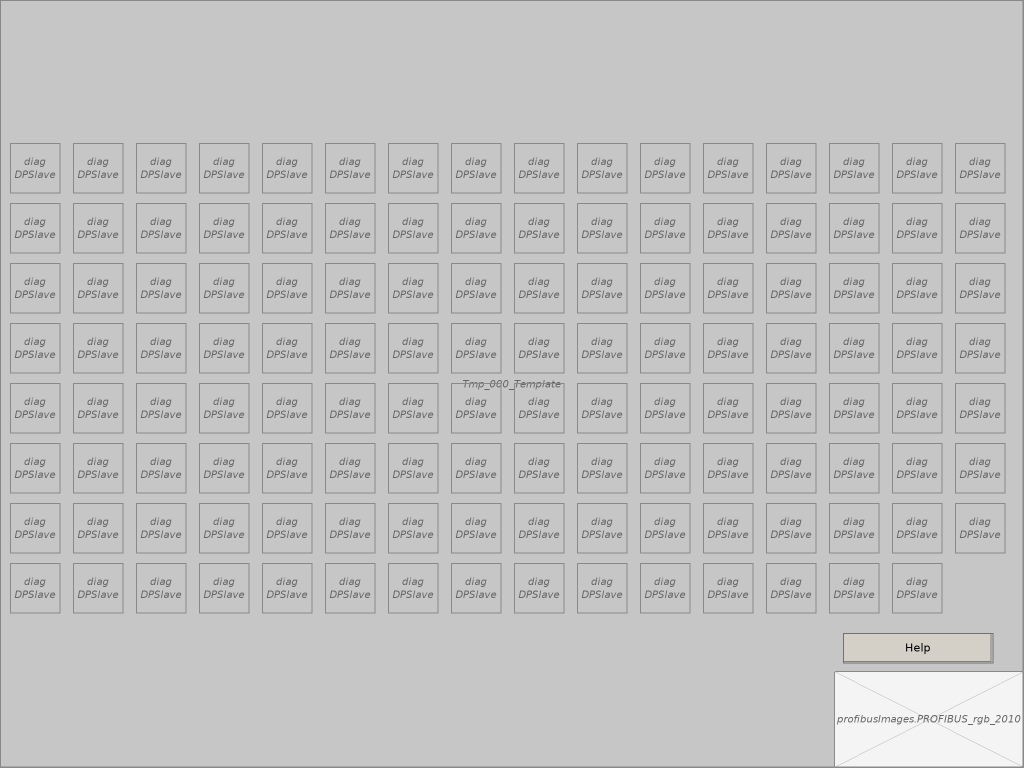
VISUALIZATION Dia_802_Profibus  // 1024x768
    Frame (0,0 1024x768)
        shows Tmp_000_Template(header := gHMIData.hmiHeader)
    Group (10,143 995x50)
        Frame (0,0 50x50)
            shows diagDPSlave(dataValues := profibusDiag.DPslaveDiag[1])
        Frame (63,0 50x50)
            shows diagDPSlave(dataValues := profibusDiag.DPslaveDiag[2])
        Frame (126,0 50x50)
            shows diagDPSlave(dataValues := profibusDiag.DPslaveDiag[3])
        Frame (189,0 50x50)
            shows diagDPSlave(dataValues := profibusDiag.DPslaveDiag[4])
        Frame (252,0 50x50)
            shows diagDPSlave(dataValues := profibusDiag.DPslaveDiag[5])
        Frame (315,0 50x50)
            shows diagDPSlave(dataValues := profibusDiag.DPslaveDiag[6])
        Frame (378,0 50x50)
            shows diagDPSlave(dataValues := profibusDiag.DPslaveDiag[7])
        Frame (441,0 50x50)
            shows diagDPSlave(dataValues := profibusDiag.DPslaveDiag[8])
        Frame (504,0 50x50)
            shows diagDPSlave(dataValues := profibusDiag.DPslaveDiag[9])
        Frame (567,0 50x50)
            shows diagDPSlave(dataValues := profibusDiag.DPslaveDiag[10])
        Frame (630,0 50x50)
            shows diagDPSlave(dataValues := profibusDiag.DPslaveDiag[11])
        Frame (693,0 50x50)
            shows diagDPSlave(dataValues := profibusDiag.DPslaveDiag[12])
        Frame (756,0 50x50)
            shows diagDPSlave(dataValues := profibusDiag.DPslaveDiag[13])
        Frame (819,0 50x50)
            shows diagDPSlave(dataValues := profibusDiag.DPslaveDiag[14])
        Frame (882,0 50x50)
            shows diagDPSlave(dataValues := profibusDiag.DPslaveDiag[15])
        Frame (945,0 50x50)
            shows diagDPSlave(dataValues := profibusDiag.DPslaveDiag[16])
    Group (10,203 995x50)
        Frame (0,0 50x50)
            shows diagDPSlave(dataValues := profibusDiag.DPslaveDiag[17])
        Frame (63,0 50x50)
            shows diagDPSlave(dataValues := profibusDiag.DPslaveDiag[18])
        Frame (126,0 50x50)
            shows diagDPSlave(dataValues := profibusDiag.DPslaveDiag[19])
        Frame (189,0 50x50)
            shows diagDPSlave(dataValues := profibusDiag.DPslaveDiag[20])
        Frame (252,0 50x50)
            shows diagDPSlave(dataValues := profibusDiag.DPslaveDiag[21])
        Frame (315,0 50x50)
            shows diagDPSlave(dataValues := profibusDiag.DPslaveDiag[22])
        Frame (378,0 50x50)
            shows diagDPSlave(dataValues := profibusDiag.DPslaveDiag[23])
        Frame (441,0 50x50)
            shows diagDPSlave(dataValues := profibusDiag.DPslaveDiag[24])
        Frame (504,0 50x50)
            shows diagDPSlave(dataValues := profibusDiag.DPslaveDiag[25])
        Frame (567,0 50x50)
            shows diagDPSlave(dataValues := profibusDiag.DPslaveDiag[26])
        Frame (630,0 50x50)
            shows diagDPSlave(dataValues := profibusDiag.DPslaveDiag[27])
        Frame (693,0 50x50)
            shows diagDPSlave(dataValues := profibusDiag.DPslaveDiag[28])
        Frame (756,0 50x50)
            shows diagDPSlave(dataValues := profibusDiag.DPslaveDiag[29])
        Frame (819,0 50x50)
            shows diagDPSlave(dataValues := profibusDiag.DPslaveDiag[30])
        Frame (882,0 50x50)
            shows diagDPSlave(dataValues := profibusDiag.DPslaveDiag[31])
        Frame (945,0 50x50)
            shows diagDPSlave(dataValues := profibusDiag.DPslaveDiag[32])
    Group (10,263 995x50)
        Frame (0,0 50x50)
            shows diagDPSlave(dataValues := profibusDiag.DPslaveDiag[33])
        Frame (63,0 50x50)
            shows diagDPSlave(dataValues := profibusDiag.DPslaveDiag[34])
        Frame (126,0 50x50)
            shows diagDPSlave(dataValues := profibusDiag.DPslaveDiag[35])
        Frame (189,0 50x50)
            shows diagDPSlave(dataValues := profibusDiag.DPslaveDiag[36])
        Frame (252,0 50x50)
            shows diagDPSlave(dataValues := profibusDiag.DPslaveDiag[37])
        Frame (315,0 50x50)
            shows diagDPSlave(dataValues := profibusDiag.DPslaveDiag[38])
        Frame (378,0 50x50)
            shows diagDPSlave(dataValues := profibusDiag.DPslaveDiag[39])
        Frame (441,0 50x50)
            shows diagDPSlave(dataValues := profibusDiag.DPslaveDiag[40])
        Frame (504,0 50x50)
            shows diagDPSlave(dataValues := profibusDiag.DPslaveDiag[41])
        Frame (567,0 50x50)
            shows diagDPSlave(dataValues := profibusDiag.DPslaveDiag[42])
        Frame (630,0 50x50)
            shows diagDPSlave(dataValues := profibusDiag.DPslaveDiag[43])
        Frame (693,0 50x50)
            shows diagDPSlave(dataValues := profibusDiag.DPslaveDiag[44])
        Frame (756,0 50x50)
            shows diagDPSlave(dataValues := profibusDiag.DPslaveDiag[45])
        Frame (819,0 50x50)
            shows diagDPSlave(dataValues := profibusDiag.DPslaveDiag[46])
        Frame (882,0 50x50)
            shows diagDPSlave(dataValues := profibusDiag.DPslaveDiag[47])
        Frame (945,0 50x50)
            shows diagDPSlave(dataValues := profibusDiag.DPslaveDiag[48])
    Group (10,323 995x50)
        Frame (0,0 50x50)
            shows diagDPSlave(dataValues := profibusDiag.DPslaveDiag[49])
        Frame (63,0 50x50)
            shows diagDPSlave(dataValues := profibusDiag.DPslaveDiag[50])
        Frame (126,0 50x50)
            shows diagDPSlave(dataValues := profibusDiag.DPslaveDiag[51])
        Frame (189,0 50x50)
            shows diagDPSlave(dataValues := profibusDiag.DPslaveDiag[52])
        Frame (252,0 50x50)
            shows diagDPSlave(dataValues := profibusDiag.DPslaveDiag[53])
        Frame (315,0 50x50)
            shows diagDPSlave(dataValues := profibusDiag.DPslaveDiag[54])
        Frame (378,0 50x50)
            shows diagDPSlave(dataValues := profibusDiag.DPslaveDiag[55])
        Frame (441,0 50x50)
            shows diagDPSlave(dataValues := profibusDiag.DPslaveDiag[56])
        Frame (504,0 50x50)
            shows diagDPSlave(dataValues := profibusDiag.DPslaveDiag[57])
        Frame (567,0 50x50)
            shows diagDPSlave(dataValues := profibusDiag.DPslaveDiag[58])
        Frame (630,0 50x50)
            shows diagDPSlave(dataValues := profibusDiag.DPslaveDiag[59])
        Frame (693,0 50x50)
            shows diagDPSlave(dataValues := profibusDiag.DPslaveDiag[60])
        Frame (756,0 50x50)
            shows diagDPSlave(dataValues := profibusDiag.DPslaveDiag[61])
        Frame (819,0 50x50)
            shows diagDPSlave(dataValues := profibusDiag.DPslaveDiag[62])
        Frame (882,0 50x50)
            shows diagDPSlave(dataValues := profibusDiag.DPslaveDiag[63])
        Frame (945,0 50x50)
            shows diagDPSlave(dataValues := profibusDiag.DPslaveDiag[64])
    Group (10,383 995x50)
        Frame (0,0 50x50)
            shows diagDPSlave(dataValues := profibusDiag.DPslaveDiag[65])
        Frame (63,0 50x50)
            shows diagDPSlave(dataValues := profibusDiag.DPslaveDiag[66])
        Frame (126,0 50x50)
            shows diagDPSlave(dataValues := profibusDiag.DPslaveDiag[67])
        Frame (189,0 50x50)
            shows diagDPSlave(dataValues := profibusDiag.DPslaveDiag[68])
        Frame (252,0 50x50)
            shows diagDPSlave(dataValues := profibusDiag.DPslaveDiag[69])
        Frame (315,0 50x50)
            shows diagDPSlave(dataValues := profibusDiag.DPslaveDiag[70])
        Frame (378,0 50x50)
            shows diagDPSlave(dataValues := profibusDiag.DPslaveDiag[71])
        Frame (441,0 50x50)
            shows diagDPSlave(dataValues := profibusDiag.DPslaveDiag[72])
        Frame (504,0 50x50)
            shows diagDPSlave(dataValues := profibusDiag.DPslaveDiag[73])
        Frame (567,0 50x50)
            shows diagDPSlave(dataValues := profibusDiag.DPslaveDiag[74])
        Frame (630,0 50x50)
            shows diagDPSlave(dataValues := profibusDiag.DPslaveDiag[75])
        Frame (693,0 50x50)
            shows diagDPSlave(dataValues := profibusDiag.DPslaveDiag[76])
        Frame (756,0 50x50)
            shows diagDPSlave(dataValues := profibusDiag.DPslaveDiag[77])
        Frame (819,0 50x50)
            shows diagDPSlave(dataValues := profibusDiag.DPslaveDiag[78])
        Frame (882,0 50x50)
            shows diagDPSlave(dataValues := profibusDiag.DPslaveDiag[79])
        Frame (945,0 50x50)
            shows diagDPSlave(dataValues := profibusDiag.DPslaveDiag[80])
    Group (10,443 995x50)
        Frame (0,0 50x50)
            shows diagDPSlave(dataValues := profibusDiag.DPslaveDiag[81])
        Frame (63,0 50x50)
            shows diagDPSlave(dataValues := profibusDiag.DPslaveDiag[82])
        Frame (126,0 50x50)
            shows diagDPSlave(dataValues := profibusDiag.DPslaveDiag[83])
        Frame (189,0 50x50)
            shows diagDPSlave(dataValues := profibusDiag.DPslaveDiag[84])
        Frame (252,0 50x50)
            shows diagDPSlave(dataValues := profibusDiag.DPslaveDiag[85])
        Frame (315,0 50x50)
            shows diagDPSlave(dataValues := profibusDiag.DPslaveDiag[86])
        Frame (378,0 50x50)
            shows diagDPSlave(dataValues := profibusDiag.DPslaveDiag[87])
        Frame (441,0 50x50)
            shows diagDPSlave(dataValues := profibusDiag.DPslaveDiag[88])
        Frame (504,0 50x50)
            shows diagDPSlave(dataValues := profibusDiag.DPslaveDiag[89])
        Frame (567,0 50x50)
            shows diagDPSlave(dataValues := profibusDiag.DPslaveDiag[90])
        Frame (630,0 50x50)
            shows diagDPSlave(dataValues := profibusDiag.DPslaveDiag[91])
        Frame (693,0 50x50)
            shows diagDPSlave(dataValues := profibusDiag.DPslaveDiag[92])
        Frame (756,0 50x50)
            shows diagDPSlave(dataValues := profibusDiag.DPslaveDiag[93])
        Frame (819,0 50x50)
            shows diagDPSlave(dataValues := profibusDiag.DPslaveDiag[94])
        Frame (882,0 50x50)
            shows diagDPSlave(dataValues := profibusDiag.DPslaveDiag[95])
        Frame (945,0 50x50)
            shows diagDPSlave(dataValues := profibusDiag.DPslaveDiag[96])
    Group (10,503 995x50)
        Frame (0,0 50x50)
            shows diagDPSlave(dataValues := profibusDiag.DPslaveDiag[97])
        Frame (63,0 50x50)
            shows diagDPSlave(dataValues := profibusDiag.DPslaveDiag[98])
        Frame (126,0 50x50)
            shows diagDPSlave(dataValues := profibusDiag.DPslaveDiag[99])
        Frame (189,0 50x50)
            shows diagDPSlave(dataValues := profibusDiag.DPslaveDiag[100])
        Frame (252,0 50x50)
            shows diagDPSlave(dataValues := profibusDiag.DPslaveDiag[101])
        Frame (315,0 50x50)
            shows diagDPSlave(dataValues := profibusDiag.DPslaveDiag[102])
        Frame (378,0 50x50)
            shows diagDPSlave(dataValues := profibusDiag.DPslaveDiag[103])
        Frame (441,0 50x50)
            shows diagDPSlave(dataValues := profibusDiag.DPslaveDiag[104])
        Frame (504,0 50x50)
            shows diagDPSlave(dataValues := profibusDiag.DPslaveDiag[105])
        Frame (567,0 50x50)
            shows diagDPSlave(dataValues := profibusDiag.DPslaveDiag[106])
        Frame (630,0 50x50)
            shows diagDPSlave(dataValues := profibusDiag.DPslaveDiag[107])
        Frame (693,0 50x50)
            shows diagDPSlave(dataValues := profibusDiag.DPslaveDiag[108])
        Frame (756,0 50x50)
            shows diagDPSlave(dataValues := profibusDiag.DPslaveDiag[109])
        Frame (819,0 50x50)
            shows diagDPSlave(dataValues := profibusDiag.DPslaveDiag[110])
        Frame (882,0 50x50)
            shows diagDPSlave(dataValues := profibusDiag.DPslaveDiag[111])
        Frame (945,0 50x50)
            shows diagDPSlave(dataValues := profibusDiag.DPslaveDiag[112])
    Frame (10,563 50x50)
        shows diagDPSlave(dataValues := profibusDiag.DPslaveDiag[113])
    Frame (73,563 50x50)
        shows diagDPSlave(dataValues := profibusDiag.DPslaveDiag[114])
    Frame (136,563 50x50)
        shows diagDPSlave(dataValues := profibusDiag.DPslaveDiag[115])
    Frame (199,563 50x50)
        shows diagDPSlave(dataValues := profibusDiag.DPslaveDiag[116])
    Frame (262,563 50x50)
        shows diagDPSlave(dataValues := profibusDiag.DPslaveDiag[117])
    Frame (325,563 50x50)
        shows diagDPSlave(dataValues := profibusDiag.DPslaveDiag[118])
    Frame (388,563 50x50)
        shows diagDPSlave(dataValues := profibusDiag.DPslaveDiag[119])
    Frame (451,563 50x50)
        shows diagDPSlave(dataValues := profibusDiag.DPslaveDiag[120])
    Frame (514,563 50x50)
        shows diagDPSlave(dataValues := profibusDiag.DPslaveDiag[121])
    Frame (577,563 50x50)
        shows diagDPSlave(dataValues := profibusDiag.DPslaveDiag[122])
    Frame (640,563 50x50)
        shows diagDPSlave(dataValues := profibusDiag.DPslaveDiag[123])
    Frame (703,563 50x50)
        shows diagDPSlave(dataValues := profibusDiag.DPslaveDiag[124])
    Frame (766,563 50x50)
        shows diagDPSlave(dataValues := profibusDiag.DPslaveDiag[125])
    Frame (829,563 50x50)
        shows diagDPSlave(dataValues := profibusDiag.DPslaveDiag[126])
    Frame (892,563 50x50)
        shows diagDPSlave(dataValues := profibusDiag.DPslaveDiag[127])
    Image (834,671 190x96), image: profibusImages.PROFIBUS_rgb_2010
    Button (843,633 150x30), "Help"
        OnMouseClick: OpenDialog Dialog=diagDPhelp, OpenModal=True, PositionX=200, PositionY=200
END_VISUALIZATION

(* stored: Version 1.1.0.1, ProductVersion 3.1.4024.12
   Visu Dia_802_Profibus: Id {b652594e-d8a5-408c-bb24-47c26b36fdb8} *)
